INTERFACE I_HydrualicPump

METHOD getSignal : BOOL
VAR_INPUT
END_VAR
END_METHOD

METHOD getState : eState
VAR_INPUT
END_VAR
END_METHOD

METHOD reset : BOOL
VAR_INPUT
END_VAR
END_METHOD

METHOD start : BOOL
VAR_INPUT
END_VAR
END_METHOD

METHOD stop : BOOL
VAR_INPUT
END_VAR
END_METHOD

END_INTERFACE

(* stored: Version 1.1.0.1, ProductVersion 3.1.4024.9
   Itf I_HydrualicPump: Id {aabcd59f-ff77-43d6-9ac8-0bc2285ce3c8}
   Method getSignal: Id {46d5db47-4070-4a63-9910-a12182a5280b}
   Method getState: Id {c9e4417b-448a-4ffe-abc9-f3ef788dfc7e}
   Method reset: Id {1dbab4cb-1482-48a3-acd7-171fec1ab50a}
   Method start: Id {f40f27b6-e1f7-4bc3-b9ce-ecba66aa1007}
   Method stop: Id {920afc6d-ae2e-4509-a1af-d878f3925590} *)
